FUNCTION_BLOCK StringBuilder IMPLEMENTS I_LimitedStringBuilder, I_StringBuilder
VAR
	sBuiltString	: T_MaxString;
END_VAR

METHOD Append : I_LimitedStringBuilder
VAR_INPUT
	sText	: T_MaxString;
END_VAR
sBuiltString := CONCAT(sBuiltString, sText);

Append := THIS^;
END_METHOD

METHOD Reset : I_LimitedStringBuilder
sBuiltString := '';

Reset := THIS^;
END_METHOD

{warning 'Add method implementation '}
METHOD ToLowerCase : I_StringBuilder
END_METHOD

METHOD ToString : T_MaxString
ToString := sBuiltString;
END_METHOD

{warning 'Add method implementation '}
METHOD ToUpperCase : I_StringBuilder
END_METHOD

END_FUNCTION_BLOCK

(* stored: Version 1.1.0.1
   POU StringBuilder: Id {669f74e3-673d-4ec6-bbfb-94c760c8d03e}, SpecialFunc None
   Method Append: Id {572aceee-1cd3-4a22-8a0a-4bfb47e5a262}
   Method Reset: Id {4dbda51d-7d32-41b5-b01c-2fef5d491479}
   Method ToLowerCase: Id {75e8326b-9ae7-4ce2-b327-2eb3e2e8b1d9}
   Method ToString: Id {aca6efb4-2aaa-4f24-83d0-e89f1255cdfd}
   Method ToUpperCase: Id {6753bb87-891c-427b-adb7-182c47965f37} *)
